// TIA Portal V20 export
DATA_BLOCK "General"   // DB2
{ S7_Optimized_Access := 'FALSE' }
AUTHOR : L.P.
// stored: AutoNumber false
   VAR RETAIN
      MEM : Struct
         off : Bool;
         on : Bool := false;
         "imp 50 ms" : Bool := false;
         "imp 100 ms" : Bool := false;
         "imp 200 ms" : Bool := false;
         "imp 400 ms" : Bool := false;
         "imp 500 ms" : Bool := false;
         "imp 800 ms" : Bool := false;
         "imp 1 s" : Bool := false;
         "imp 1,6 s" : Bool := false;
         "imp 2 s" : Bool := false;
         "HM imp 50 ms 1" : Bool := false;
         "HM imp 50 ms 2" : Bool := false;
         "HM imp 100 ms" : Bool := false;
         "HM imp 200 ms" : Bool := false;
         "HM imp 400 ms" : Bool := false;
         "HM imp 500 ms" : Bool := false;
         "HM imp 800 ms" : Bool := false;
         "HM imp 1 s" : Bool := false;
         "HM imp 1,6 s" : Bool := false;
         "HM imp 2 s" : Bool := false;
         "single pal" : Bool := false;
         "douple pal" : Bool := false;
         "warm start" : Bool := false;
         commissioning : Bool := false;
         "pal is model M5" : Bool;
         "pal is model M6" : Bool := false;
         "pal is model M7" : Bool := false;
         "29" : Bool := false;
         "pal is model M9" : Bool := false;
         "31" : Bool := false;
         "32" : Bool := false;
         "33" : Bool := false;
         "34" : Bool := false;
         "35" : Bool := false;
         "pal with stacker" : Bool := false;
         "37" : Bool := false;
         "38" : Bool := false;
         "39" : Bool := false;
         "pal with single infeed" : Bool := false;
         "pal with double infeed" : Bool := false;
         "42" : Bool := false;
         "43" : Bool := false;
         "stop cycle with button" : Bool := false;
         "drive RLP in safe position in stop cycle" : Bool := false;
         "46" : Bool := false;
         "47" : Bool := false;
         "48" : Bool := false;
         "49" : Bool := false;
         "wrapper with film clamp above" : Bool := false;
         "wrapper with film clamp on carriage" : Bool := false;
         "52" : Bool := false;
         "53" : Bool := false;
         "54" : Bool := false;
         "55" : Bool := false;
         "56" : Bool := false;
         "57" : Bool := false;
         "58" : Bool := false;
         "59" : Bool := false;
         "60" : Bool := false;
         "61" : Bool := false;
         "62" : Bool := false;
         "63" : Bool := false;
         "64" : Bool := false;
         "65" : Bool := false;
         "66" : Bool := false;
         "67" : Bool := false;
         "68" : Bool := false;
         "69" : Bool := false;
         "70" : Bool := false;
         "71" : Bool := false;
         "72" : Bool := false;
         "73" : Bool := false;
         "74" : Bool := false;
         "75" : Bool := false;
         "76" : Bool := false;
         "77" : Bool := false;
         "78" : Bool := false;
         "79" : Bool := false;
         "80" : Bool := false;
         "81" : Bool := false;
         "82" : Bool := false;
         "83" : Bool := false;
         "84" : Bool := false;
         "85" : Bool := false;
         "86" : Bool := false;
         "87" : Bool := false;
         "88" : Bool := false;
         "89" : Bool := false;
         "90" : Bool := false;
         "91" : Bool := false;
         "92" : Bool := false;
         "93" : Bool := false;
         "94" : Bool := false;
         "95" : Bool := false;
         "96" : Bool := false;
         "97" : Bool := false;
         "98" : Bool := false;
         "99" : Bool := false;
         "100" : Bool := false;
      END_STRUCT;
      "STEP" : Struct
         "0" : Bool;
         "1" : Bool;
         "2" : Bool := false;
         "3" : Bool := false;
         "4" : Bool := false;
         "5" : Bool := false;
         "6" : Bool := false;
         "7" : Bool := false;
         "8" : Bool := false;
         "9" : Bool := false;
         "10" : Bool := false;
      END_STRUCT;
      T : Struct
         "delay wachdog to FEE" { S7_SetPoint := 'True'} : IEC_TIMER;
         "delay no conection to FEE" { S7_SetPoint := 'True'} : IEC_TIMER;
         "3" { S7_SetPoint := 'True'} : IEC_TIMER;
         "4" { S7_SetPoint := 'True'} : IEC_TIMER;
         "5" { S7_SetPoint := 'True'} : IEC_TIMER;
         "6" { S7_SetPoint := 'True'} : IEC_TIMER;
         "7" { S7_SetPoint := 'True'} : IEC_TIMER;
         "8" { S7_SetPoint := 'True'} : IEC_TIMER;
         "9" { S7_SetPoint := 'True'} : IEC_TIMER;
         "10" { S7_SetPoint := 'True'} : IEC_TIMER;
         "11" { S7_SetPoint := 'True'} : IEC_TIMER;
         "12" { S7_SetPoint := 'True'} : IEC_TIMER;
         "13" { S7_SetPoint := 'True'} : IEC_TIMER;
         "14" { S7_SetPoint := 'True'} : IEC_TIMER;
         "15" { S7_SetPoint := 'True'} : IEC_TIMER;
         "16" { S7_SetPoint := 'True'} : IEC_TIMER;
         "17" { S7_SetPoint := 'True'} : IEC_TIMER;
         "18" { S7_SetPoint := 'True'} : IEC_TIMER;
         "19" { S7_SetPoint := 'True'} : IEC_TIMER;
         "20" { S7_SetPoint := 'True'} : IEC_TIMER;
         "21" { S7_SetPoint := 'True'} : IEC_TIMER;
         "22" { S7_SetPoint := 'True'} : IEC_TIMER;
         "23" { S7_SetPoint := 'True'} : IEC_TIMER;
         "24" { S7_SetPoint := 'True'} : IEC_TIMER;
         "25" { S7_SetPoint := 'True'} : IEC_TIMER;
         "26" { S7_SetPoint := 'True'} : IEC_TIMER;
         "27" { S7_SetPoint := 'True'} : IEC_TIMER;
         "28" { S7_SetPoint := 'True'} : IEC_TIMER;
         "29" { S7_SetPoint := 'True'} : IEC_TIMER;
         "30" { S7_SetPoint := 'True'} : IEC_TIMER;
      END_STRUCT;
      C : Struct
         "1" { S7_SetPoint := 'True'} : IEC_COUNTER;
         "2" { S7_SetPoint := 'True'} : IEC_COUNTER;
         "3" { S7_SetPoint := 'True'} : IEC_COUNTER;
         "4" { S7_SetPoint := 'True'} : IEC_COUNTER;
         "5" { S7_SetPoint := 'True'} : IEC_COUNTER;
         "6" { S7_SetPoint := 'True'} : IEC_COUNTER;
         "7" { S7_SetPoint := 'True'} : IEC_COUNTER;
         "8" { S7_SetPoint := 'True'} : IEC_COUNTER;
         "9" { S7_SetPoint := 'True'} : IEC_COUNTER;
         "10" { S7_SetPoint := 'True'} : IEC_COUNTER;
         "11" { S7_SetPoint := 'True'} : IEC_COUNTER;
         "12" { S7_SetPoint := 'True'} : IEC_COUNTER;
         "13" { S7_SetPoint := 'True'} : IEC_COUNTER;
         "14" { S7_SetPoint := 'True'} : IEC_COUNTER;
         "15" { S7_SetPoint := 'True'} : IEC_COUNTER;
         "16" { S7_SetPoint := 'True'} : IEC_COUNTER;
         "17" { S7_SetPoint := 'True'} : IEC_COUNTER;
         "18" { S7_SetPoint := 'True'} : IEC_COUNTER;
         "19" { S7_SetPoint := 'True'} : IEC_COUNTER;
         "20" { S7_SetPoint := 'True'} : IEC_COUNTER;
         "21" { S7_SetPoint := 'True'} : IEC_COUNTER;
         "22" { S7_SetPoint := 'True'} : IEC_COUNTER;
         "23" { S7_SetPoint := 'True'} : IEC_COUNTER;
         "24" { S7_SetPoint := 'True'} : IEC_COUNTER;
         "25" { S7_SetPoint := 'True'} : IEC_COUNTER;
         "26" { S7_SetPoint := 'True'} : IEC_COUNTER;
         "27" { S7_SetPoint := 'True'} : IEC_COUNTER;
         "28" { S7_SetPoint := 'True'} : IEC_COUNTER;
         "29" { S7_SetPoint := 'True'} : IEC_COUNTER;
         "30" { S7_SetPoint := 'True'} : IEC_COUNTER;
      END_STRUCT;
      DATA : Struct
         Byte1 : Byte;
         Byte2 : Byte := 16#0;
         Byte3 : Byte := 16#0;
         Byte4 : Byte := 16#0;
         Byte5 : Byte := 16#0;
         Byte6 : Byte := 16#0;
         Byte7 : Byte := 16#0;
         Byte8 : Byte := 16#0;
         Byte9 : Byte := 16#0;
         Byte10 : Byte := 16#0;
         "PAL NR" : Int;
         "Buffer Watchdog FEE" : Int;
         Int3 : Int := 0;
         Int4 : Int := 0;
         Int5 : Int := 0;
         Int6 : Int := 0;
         Int7 : Int;
         Int8 : Int := 0;
         Int9 : Int;
         Int10 : Int := 0;
         Dint1 : DInt;
         Dint2 : DInt := 0;
         Dint3 : DInt;
         Dint4 : DInt := 0;
         Dint5 : DInt;
         Dint6 : DInt := 0;
         Dint7 : DInt := 0;
         Dint8 : DInt := 0;
         Dint9 : DInt := 0;
         Dint10 : DInt := 0;
         "screen number HMI" : Array[0..4] of Int;
      END_STRUCT;
   END_VAR
BEGIN
END_DATA_BLOCK
